TYPE Read_INJLPS_Values_To_PC_Struct :
UNION
	S_INJLPSValues_To_PC:S_INJLPSValues_To_PC_Struct;
END_UNION
END_TYPE

(* stored: Version 1.1.0.1, ProductVersion 3.1.4024.16
   DUT Read_INJLPS_Values_To_PC_Struct: Id {94145265-0621-4840-a36d-7bc2a30f5281} *)
